// TIA Portal project "BurnerAlarm_LAD" (V17)

(* hardware
DEVICE "PLC_1"  S7-1200 Station
   slot 0: "Rack_0"  S7-1200 Rack  Rack  V1.0
   slot 1: "PLC_1"  CPU 1214C AC/DC/Rly  6ES7 214-1BG40-0XB0  V4.5
*)

// ===== PLC "PLC_1"  CPU 1214C AC/DC/Rly =====

VAR_GLOBAL   // PLC tag table "烧嘴报警变量表"
   "1#故障反馈" AT %I0.1 : Bool;
   "2#故障反馈" AT %I0.4 : Bool;
   "3#故障反馈" AT %I0.7 : Bool;
   "4#故障反馈" AT %I1.2 : Bool;
   "5#故障反馈" AT %I1.5 : Bool;
   "6#故障反馈" AT %I2.2 : Bool;
   "7#故障反馈" AT %I2.5 : Bool;
   "蜂鸣器" AT %Q4.7 : Bool;
END_VAR

DATA_BLOCK "内部数据"   // DB1
{ S7_Optimized_Access := 'TRUE' }
VERSION : 0.1
   VAR
      报警脉冲 : Bool;   // P_TRIG上升沿存储位
      控温超温标志 : Bool;   // 任意一区超温汇总标志
   END_VAR
BEGIN
END_DATA_BLOCK

DATA_BLOCK "数字量信号"   // DB2
{ S7_Optimized_Access := 'TRUE' }
VERSION : 0.1
   VAR
      超温标志_1区 : Bool;   // 1区超温
      超温标志_2区 : Bool;   // 2区超温
      超温标志_3区 : Bool;   // 3区超温
      超温标志_4区 : Bool;   // 4区超温
      超温标志_5区 : Bool;   // 5区超温
      超温标志_6区 : Bool;   // 6区超温
   END_VAR
BEGIN
END_DATA_BLOCK

FUNCTION "FC_BurnerAlarm" : Void   // FC1, LAD
{ S7_Optimized_Access := 'TRUE' }
   VAR_TEMP   // added for the SCL form of the ladder/FBD networks
      _w1 : Bool;
      _w2 : Bool;
   END_VAR
BEGIN

REGION Network 1: 烧嘴故障报警置位蜂鸣器
   // 七个烧嘴故障反馈常开触点并联，汇总信号接入P_TRIG上升沿检测，任意故障反馈上升沿置位蜂鸣器输出。
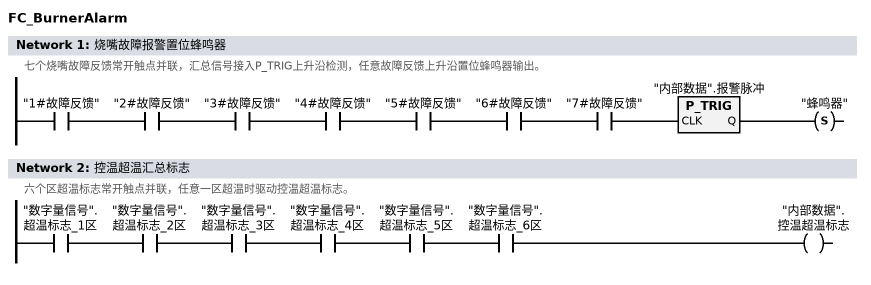
   RUNG wire#powerrail
      Contact( "1#故障反馈" )
      Contact( "2#故障反馈" )
      Contact( "3#故障反馈" )
      Contact( "4#故障反馈" )
      Contact( "5#故障反馈" )
      Contact( "6#故障反馈" )
      Contact( "7#故障反馈" )
      P_Trig( "内部数据".报警脉冲 )
      S_Coil( "蜂鸣器" )
   END_RUNG
   // the same network as SCL:
   #_w1 := "1#故障反馈" AND "2#故障反馈" AND "3#故障反馈" AND "4#故障反馈" AND "5#故障反馈" AND "6#故障反馈" AND "7#故障反馈";
   #_w2 := #_w1 AND NOT "内部数据".报警脉冲;   // rising edge
   "内部数据".报警脉冲 := #_w1;
   IF #_w2 THEN "蜂鸣器" := TRUE; END_IF;
END_REGION

REGION Network 2: 控温超温汇总标志
   // 六个区超温标志常开触点并联，任意一区超温时驱动控温超温标志。
   RUNG wire#powerrail
      Contact( "数字量信号".超温标志_1区 )
      Contact( "数字量信号".超温标志_2区 )
      Contact( "数字量信号".超温标志_3区 )
      Contact( "数字量信号".超温标志_4区 )
      Contact( "数字量信号".超温标志_5区 )
      Contact( "数字量信号".超温标志_6区 )
      Coil( "内部数据".控温超温标志 )
   END_RUNG
   // the same network as SCL:
   "内部数据".控温超温标志 := "数字量信号".超温标志_1区 AND "数字量信号".超温标志_2区 AND "数字量信号".超温标志_3区 AND "数字量信号".超温标志_4区 AND "数字量信号".超温标志_5区 AND "数字量信号".超温标志_6区;
END_REGION
END_FUNCTION

ORGANIZATION_BLOCK "Main"   // OB1, LAD, ProgramCycle
TITLE = "Main Program Sweep (Cycle)"
{ S7_Optimized_Access := 'TRUE' }
VERSION : 0.1
   VAR_INPUT
      Initial_Call : Bool;   // Initial call of this OB
      Remanence : Bool;   // =True, if remanent data are available
   END_VAR
BEGIN
END_ORGANIZATION_BLOCK